PROGRAM P_Startup
VAR
	bDone	: BOOL;
END_VAR

IF NOT bDone THEN
	GVL_System.fbStation.Reset();
	GVL_System.fbDerived.Reset();
	GVL_Hmi.nSpeed := 50;
	bDone := TRUE;
END_IF

END_PROGRAM

(* stored: Version 1.1.0.1, ProductVersion 3.1.4024.12
   POU P_Startup: Id {fb1714d1-1e4d-4ffd-9865-7a2e3d94ba82}, SpecialFunc None *)
